FUNCTION_BLOCK getSDOMotorErrorFlags
VAR_INPUT
	nSlaveAddr: UINT;
	nIndex: WORD;
END_VAR

VAR_OUTPUT
	Overtemp: BOOL;
	Torqueoverload: BOOL;
	Shortcircuit: BOOL;
	
END_VAR
VAR

	Short_CircuitBlock: FB_EcCoESdoRead;
	Torque_OverloadBlock: FB_EcCoESdoRead;
	Over_TemperatureBlock: FB_EcCoESdoRead;

	trigger: BOOL;
	TON_0: TON;
	TON_1: TON;
	ms: TIME;

END_VAR

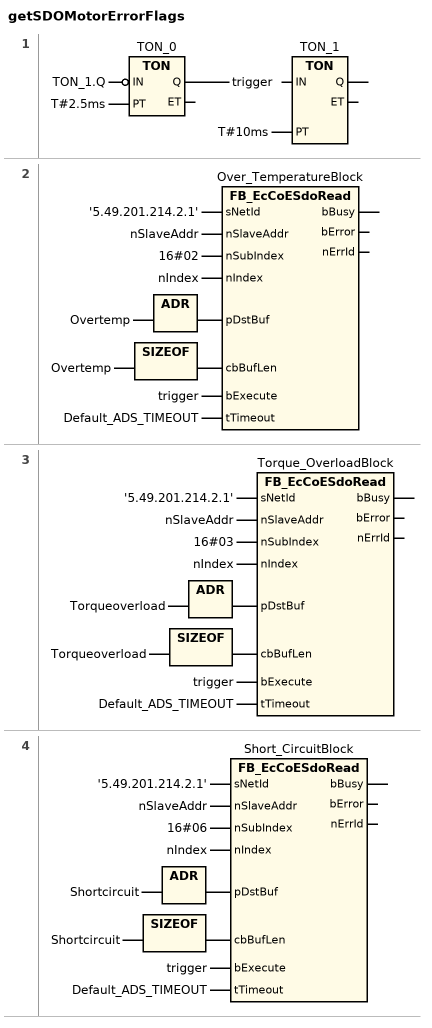
// NETWORK 1
TON_0(IN := NOT TON_1.Q, PT := T#2.5ms); // TON
trigger := TON_0.Q;
TON_1(IN := TON_0.Q, PT := T#10ms); // TON

// NETWORK 2
Over_TemperatureBlock(
    sNetId := '5.49.201.214.2.1',
    nSlaveAddr := nSlaveAddr,
    nSubIndex := 16#02,
    nIndex := nIndex,
    pDstBuf := ADR(Overtemp),
    cbBufLen := SIZEOF(Overtemp),
    bExecute := trigger,
    tTimeout := Default_ADS_TIMEOUT); // FB_EcCoESdoRead

// NETWORK 3
Torque_OverloadBlock(
    sNetId := '5.49.201.214.2.1',
    nSlaveAddr := nSlaveAddr,
    nSubIndex := 16#03,
    nIndex := nIndex,
    pDstBuf := ADR(Torqueoverload),
    cbBufLen := SIZEOF(Torqueoverload),
    bExecute := trigger,
    tTimeout := Default_ADS_TIMEOUT); // FB_EcCoESdoRead

// NETWORK 4
Short_CircuitBlock(
    sNetId := '5.49.201.214.2.1',
    nSlaveAddr := nSlaveAddr,
    nSubIndex := 16#06,
    nIndex := nIndex,
    pDstBuf := ADR(Shortcircuit),
    cbBufLen := SIZEOF(Shortcircuit),
    bExecute := trigger,
    tTimeout := Default_ADS_TIMEOUT); // FB_EcCoESdoRead

END_FUNCTION_BLOCK

(* stored: Version 1.1.0.1, ProductVersion 3.1.4022.3
   POU getSDOMotorErrorFlags: Id {d3f3239f-12eb-4abb-a467-1c39e123c318}, SpecialFunc None *)
